# EPICS substitutions: ethmodApp/Db/AKI2C_M24M02.substitutions
file AKI2C_M24M02_dev.template
{
   pattern { P    ,R    ,PORT    ,ADDR     ,TIMEOUT     }
           { $(P) ,$(R) ,$(PORT) ,$(ADDR)  ,$(TIMEOUT)  }
}
